TYPE HaProduct :
STRUCT
	name			:	STRING;
	identifiers		:	ARRAY[1..1] OF STRING := ['smart dims'];
	model			:	STRING;
	manufacturer	:	STRING;
END_STRUCT
END_TYPE

(* stored: Version 1.1.0.1, ProductVersion 3.1.4024.12
   DUT HaProduct: Id {1ca5529f-320b-4d0d-b0ac-b65869999385} *)
